TYPE ST_Timedata_2 :
STRUCT
	
	RunTime:ARRAY[0..25] OF UINT;//运行时间
    WaitTime:ARRAY[0..25] OF UINT;//待机时间
    AlmTime:ARRAY[0..25] OF UINT;//报警时间 	
    changeTime:ARRAY[0..25] OF UINT;//极片更换等待时间  	

	
END_STRUCT
END_TYPE

(* stored: Version 1.1.0.1, ProductVersion 3.1.4024.9
   DUT ST_Timedata_2: Id {36e775a0-6569-4c9b-980c-5e4ac9c2a167} *)
